(* Logix 5000 project; controller ktc_lab2 vendor 1 type 14 code 150 rev 30.11; software revision 30.00 *)

TASK MainTask (continuous, watchdog 500 ms) : MainProgram

MODULES
   Local : vendor 1 type 14 code 150 (Compact 0, rev 30.11)
      Counters : Embedded (Compact 3, rev 1.1, Output RPI 20 ms)
      Discrete_IO : Embedded (Compact 1, rev 3.1, Output RPI 20 ms)
      Analog_IO : Embedded (Compact 2, rev 1.1, Output RPI 80 ms)
END_MODULES

PROGRAM MainProgram   (* main routine MainRoutine *)
VAR
   M1 : ALIAS FOR Local:1:O.Data.1;   // MOTOR
   M6 : ALIAS FOR Local:1:O.Data.6;   // PL6 MOTOR
   PB1 : ALIAS FOR Local:1:I.Data.1;   // START
   PB2 : ALIAS FOR Local:1:I.Data.3;   // STOP PBNC
   PB3 : ALIAS FOR Local:1:I.Data.0;   // START
   PB4 : ALIAS FOR Local:1:I.Data.2;   // STOP PBNC
   pl1 : BOOL;
   pl1_2 : BOOL;
   pl1_3 : BOOL := 1;
   PL1B : ALIAS FOR Local:1:O.Data.3;   // CAUTION
   pl2 : BOOL;
   pl2_2 : BOOL;
   pl2_3 : BOOL;
   pl3_2 : BOOL := 1;
   pl3_3 : BOOL;
   pl4_2 : BOOL := 1;
   pl4_3 : BOOL := 1;
   PL4C : ALIAS FOR Local:1:O.Data.2;
   PL5C : ALIAS FOR Local:1:O.Data.0;   // MOTOR LIGHT
   sw1 : BOOL := 1;
   sw2 : BOOL;
   sw3 : BOOL;
   sw4 : BOOL;
   sw5 : BOOL := 1;
   sw6 : BOOL;
   T4_1 : TIMER := (PRE := 10000);
   T4_2 : TIMER := (PRE := 5000);
   T4_3 : TIMER := (PRE := 1000);
   T4_4 : TIMER := (PRE := 500);
   T4_5 : TIMER := (PRE := 5000);
   T4_6 : TIMER := (PRE := 500);
   T4_7 : TIMER := (PRE := 1000);
   T4_8 : TIMER := (PRE := 500);
   T4_9 : TIMER := (PRE := 1000);
END_VAR

ROUTINE MainRoutine   (* ladder *)
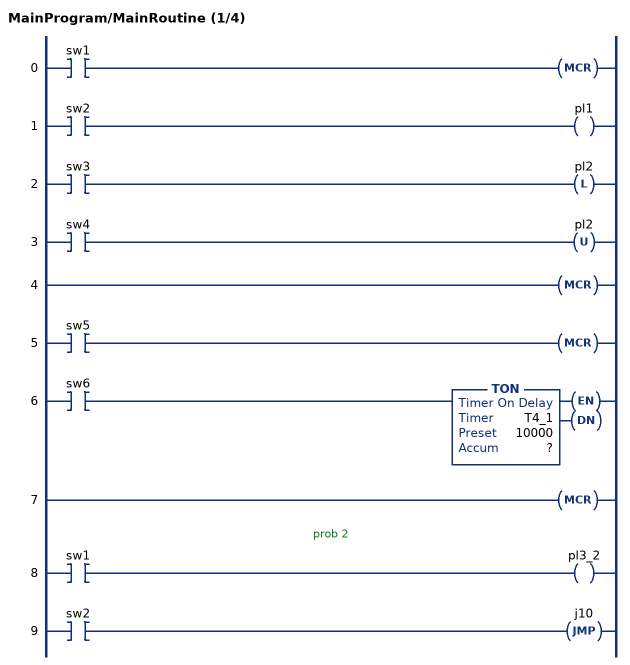
   0: XIC(sw1)MCR();
   1: XIC(sw2)OTE(pl1);
   2: XIC(sw3)OTL(pl2);
   3: XIC(sw4)OTU(pl2);
   4: MCR();
   5: XIC(sw5)MCR();
   6: XIC(sw6)TON(T4_1,?,?);
   7: MCR();
   // prob 2
   8: XIC(sw1)OTE(pl3_2);
   9: XIC(sw2)JMP(j10);
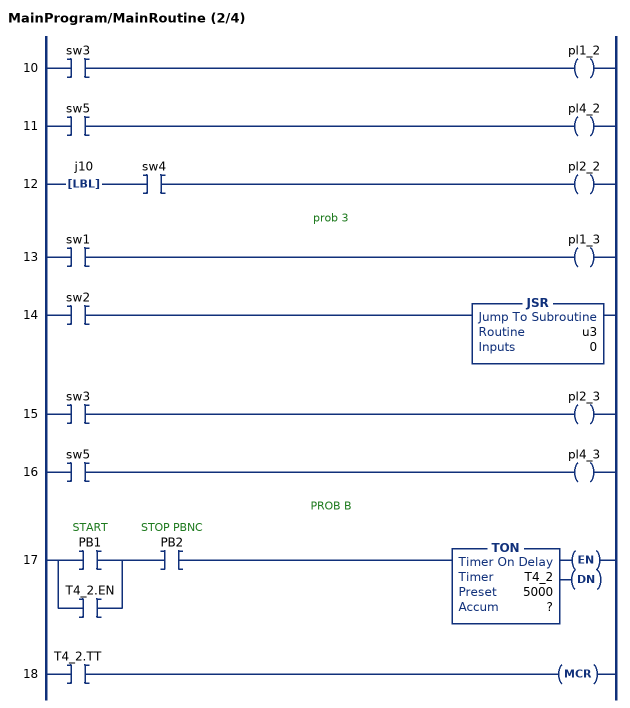
   10: XIC(sw3)OTE(pl1_2);
   11: XIC(sw5)OTE(pl4_2);
   12: LBL(j10)XIC(sw4)OTE(pl2_2);
   // prob 3
   13: XIC(sw1)OTE(pl1_3);
   14: XIC(sw2)JSR(u3,0);
   15: XIC(sw3)OTE(pl2_3);
   16: XIC(sw5)OTE(pl4_3);
   // PROB B
   17: [XIC(PB1) ,XIC(T4_2.EN) ]XIC(PB2)TON(T4_2,?,?);
   18: XIC(T4_2.TT)MCR();
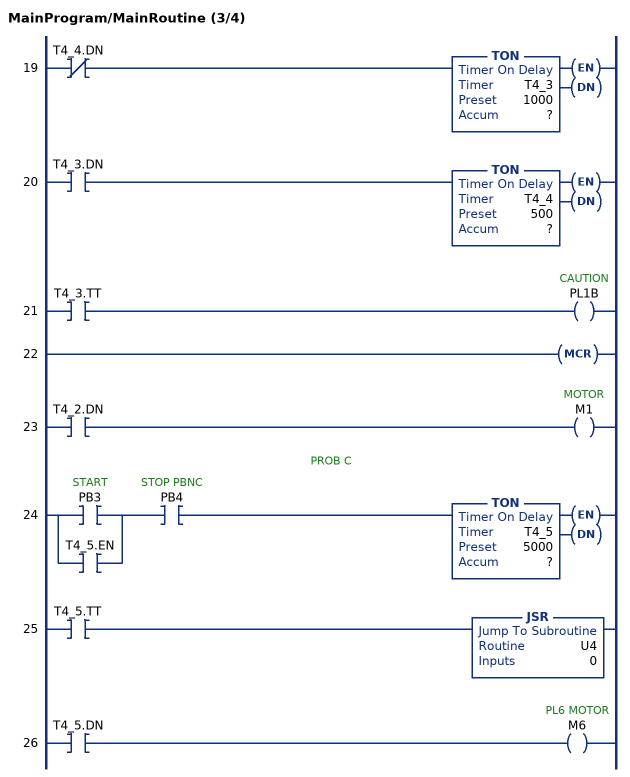
   19: XIO(T4_4.DN)TON(T4_3,?,?);
   20: XIC(T4_3.DN)TON(T4_4,?,?);
   21: XIC(T4_3.TT)OTE(PL1B);
   22: MCR();
   23: XIC(T4_2.DN)OTE(M1);
   // PROB C
   24: [XIC(PB3) ,XIC(T4_5.EN) ]XIC(PB4)TON(T4_5,?,?);
   25: XIC(T4_5.TT)JSR(U4,0);
   26: XIC(T4_5.DN)OTE(M6);
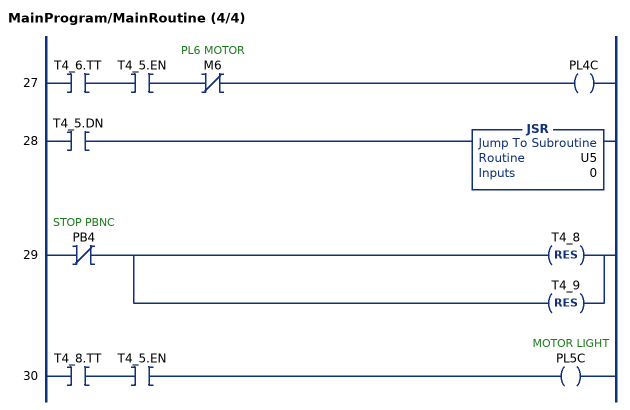
   27: XIC(T4_6.TT)XIC(T4_5.EN)XIO(M6)OTE(PL4C);
   28: XIC(T4_5.DN)JSR(U5,0);
   29: XIO(PB4)[RES(T4_8) ,RES(T4_9) ];
   30: XIC(T4_8.TT)XIC(T4_5.EN)OTE(PL5C);
END_ROUTINE

ROUTINE u3   (* ladder *)
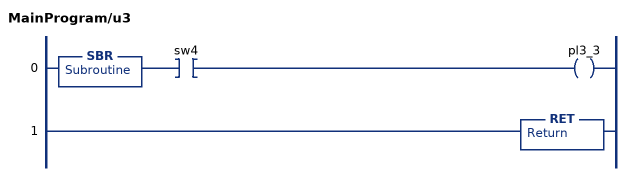
   0: SBR()XIC(sw4)OTE(pl3_3);
   1: RET();
END_ROUTINE

ROUTINE U4   (* ladder *)
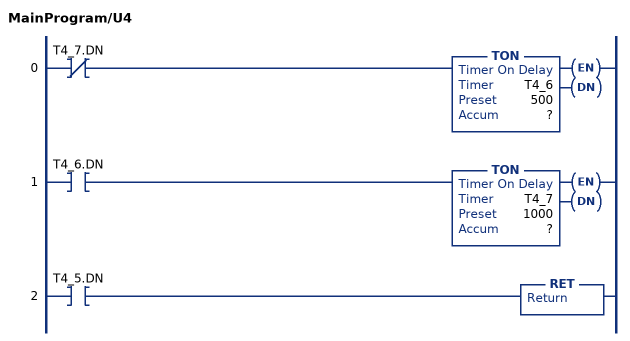
   0: XIO(T4_7.DN)TON(T4_6,?,?);
   1: XIC(T4_6.DN)TON(T4_7,?,?);
   2: XIC(T4_5.DN)RET();
END_ROUTINE

ROUTINE U5   (* ladder *)
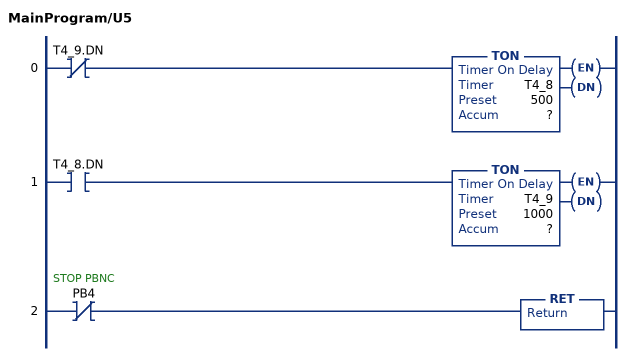
   0: XIO(T4_9.DN)TON(T4_8,?,?);
   1: XIC(T4_8.DN)TON(T4_9,?,?);
   2: XIO(PB4)RET();
END_ROUTINE
END_PROGRAM
